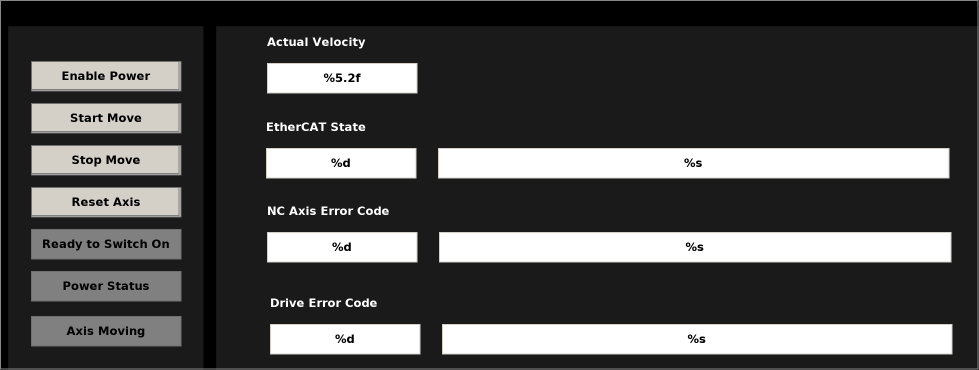
VISUALIZATION Visualization  // 979x370
    Rectangle (216,26 763x344)
    Rectangle (8,26 195x344)
    Button (31,61 150x30), "Enable Power", colour toggle: MAIN.enable_power
        toggle MAIN.enable_power
    Button (31,103 150x30), "Start Move"
        tap MAIN.enable_move
    Button (31,145 150x30), "Stop Move"
        tap MAIN.enable_stop
    Button (31,187 150x30), "Reset Axis"
        tap MAIN.enable_reset
    Textfield (438,148 511x30), "%s", text variable: MAIN.Ax8206_ChA_Decoder.sDriveEcState
    Textfield (266,148 150x30), "%d", text variable: MAIN.Ax8206_ChA_Decoder.nDriveEcState
    Label (263,112 215x30), "EtherCAT State"
    Textfield (267,63 150x30), "%5.2f", text variable: MAIN.Ax8206_ChA_Ref.NcToPlc.ActVelo
    Label (264,27 215x30), "Actual Velocity"
    Button (31,229 150x30), "Ready to Switch On", colour toggle: MAIN.Ax8206_ChA_Decoder.nDSP402status.0
    Button (31,316 150x30), "Axis Moving", colour toggle: MAIN.Ax8206_ChA_Ref.Status.Moving
    Textfield (439,232 512x30), "%s", text variable: MAIN.Ax8206_ChA_Decoder.sNcError
    Textfield (267,232 150x30), "%d", text variable: MAIN.Ax8206_ChA_Decoder.nNcError
    Label (264,196 215x30), "NC Axis Error Code"
    Textfield (442,324 510x30), "%s", text variable: MAIN.Ax8206_ChA_Decoder.sDriveError
    Textfield (270,324 150x30), "%d", text variable: MAIN.Ax8206_ChA_Decoder.nDriveError
    Label (267,288 215x30), "Drive Error Code"
    Button (31,271 150x30), "Power Status", colour toggle: MAIN.fb_power.Status
END_VISUALIZATION

(* stored: Version 1.1.0.1, ProductVersion 3.1.4024.12
   Visu Visualization: Id {a9f69750-988d-044f-1def-8bdeadd3b27e} *)
